TYPE "SpeedMachine_COut"
VERSION : 0.1
// Block: SpeedMachine_COut
   STRUCT
      Infeed_ReqON : Bool;
      CtrlSafe : Bool;
      Standstill : Bool;
      Bwd_CheckNext : Bool;
      Fwd_CheckNext : Bool;
      Bwd_VelZero : Bool;
      Bwd_Running : Bool;
      Fwd_VelZero : Bool;
      Fwd_Running : Bool;
      ActualVelocity : LReal;
      TargetVelocity : LReal;
      MaxVelocity : LReal;
   END_STRUCT;

END_TYPE
